{attribute 'qualified_only'}
VAR_GLOBAL CONSTANT
	nSubUnits	:	UINT		:=	1;
	
END_VAR

(* stored: Version 1.1.0.1, ProductVersion 3.1.4022.16
   GVL CONST_GV: Id {20b675dd-a58e-40bd-8118-f7a208e47392} *)
